// TIA Portal V19 export
FUNCTION_BLOCK "TYPIC_C403_SF_LVE"   // FB131, FBD
TITLE = TYPIC_C403_SF_LVE: Detectiepunt
{ S7_Optimized_Access := 'TRUE' }
AUTHOR : OCOTECH
FAMILY : Typical
NAME : C403.802
// Logisch Object Besturing: C403.802
// 
// De subfunctie detectiepunt verzorgt de bediening en sturing van een SOSodetectiepunt vanuit 3B en is tevens het raakvlak tussen 3B en de interne sturing van het detectiepunt.
// stored: MemoryReserve 10, SetENOAutomatically false
   VAR_INPUT
      CFG_STR { ExternalAccessible := 'False'; ExternalVisible := 'False'; ExternalWritable := 'False'} : USInt;   // Nummer van de rijstrook (1 = rechterrijstrook)
      CFG_NUM { ExternalAccessible := 'False'; ExternalVisible := 'False'; ExternalWritable := 'False'} : Int;   // Nummer van het detectiepunt op de rijstrook volgens rijrichting
      CFG_POS1 { ExternalAccessible := 'False'; ExternalVisible := 'False'; ExternalWritable := 'False'} : USInt;   // FO-naam van de verkeerskoker (of op- / afrit) waar het detectiepunt staat
      CFG_POS2 { ExternalAccessible := 'False'; ExternalVisible := 'False'; ExternalWritable := 'False'} : Real;   // Lengtepositie van het detectiepunt in de verkeerskoker
      CFG_LCK_AANT { ExternalAccessible := 'False'; ExternalVisible := 'False'; ExternalWritable := 'False'} : Int;   // Aantal stroomopwaartse detectiepunten waarin verkeerskundige meldingen onderdrukt worden
      STU_ALG_LCK_SIG { ExternalAccessible := 'False'; ExternalVisible := 'False'; ExternalWritable := 'False'} : USInt;   // Onderdruk alarmen
   END_VAR
   VAR_OUTPUT
      VAR_LVE { ExternalAccessible := 'False'; ExternalVisible := 'False'; ExternalWritable := 'False'} : "C403_VAR_LVE_TYPIC";   // Struct met alle variabelen van de SOS-sectie
   END_VAR
   VAR_IN_OUT
      STU_LVE : "C403_STU_LVE_TYPIC";   // Sturing Detectiepunten
      VAR_IF_LVE : "C403_VAR_IF_LVE_TYPIC";   // Struct met alle variabelen ontvangen van de functie (IF) in de interne sturing van het afsluitsysteem
   END_VAR
   VAR
      BED : Struct   // Bedieningen
         OBS : Struct   // SOS-sectie aan- of uitschakelen
            X : "UDT_BED_ALG";
            KNOP { S7_SetPoint := 'True'} : Array[0..1] of "UDT_BED_KNOP";
         END_STRUCT;
         VGV_SIG : Struct   // Signalering verkeerskundige alarmen vrijgeven of onderdrukken
            X : "UDT_BED_ALG";
            KNOP { S7_SetPoint := 'True'} : Array[0..1] of "UDT_BED_KNOP";
         END_STRUCT;
      END_STRUCT;
      BED_OBS { ExternalWritable := 'False'} : "TYPIC_HF_BED_ALG_KNOP";   // SOS-sectie aan- of uitschakelen
      BED_VGV_SIG { ExternalWritable := 'False'} : "TYPIC_HF_BED_ALG_KNOP";   // Signalering verkeerskundige alarmen vrijgeven of onderdrukken
      SIG { ExternalWritable := 'False'} : Struct   // Signaleringen
         AA01 : Bool;   // Detectiepunt niet observeerbaar
         AA02 : Bool;   // Storing algemeen
         AA03 : Bool;   // Deur wegkantkast geopend
         AV01 : Bool;   // Stilstand gedetecteerd
         AV02 : Bool;   // Snelheidsonderschrijding gedetecteerd
         AV03 : Bool;   // Spookrijder gedetecteerd
         A001 : Bool;   // Beveiliging aangesproken
         A002 : Bool;   // Storing detectiepunt
         A003 : Bool;   // Beveiliging klimaatregeling wegkantkast aangesproken
         A004 : Bool;   // Overspanningsbeveiliging aangesproken
      END_STRUCT;
      VAR { ExternalWritable := 'False'} : Struct   // Variabelen
         STS_STOP : USInt;   // Stilstand gedetecteerd
         STS_SOS : USInt;   // Snelheidsonderschrijding gedetecteerd
         RNO : USInt;   // Reden niet bestuurbaar
         VGV_SIG_VOP : Bool;   // TRUE = Signaleringen vrijgegeven voor verkeersoperator FALSE = Onderdrukt
         MEM_STS_STOP { ExternalAccessible := 'False'; ExternalVisible := 'False'} : Bool;   // TRUE = Stilstand gedetecteerd
         MEM_STS_SOS { ExternalAccessible := 'False'; ExternalVisible := 'False'} : Bool;   // TRUE = Snelheidsonderschrijding gedetecteerd
         STS_STOP_NEW { ExternalAccessible := 'False'; ExternalVisible := 'False'} : Bool;   // TRUE = Nieuwe detectie Stilstand
         STS_SOS_NEW { ExternalAccessible := 'False'; ExternalVisible := 'False'} : Bool;   // TRUE = Nieuwe detectie snelheidsonderschrijding
         LCK_STOP { ExternalAccessible := 'False'; ExternalVisible := 'False'} : Bool;   // TRUE = Onderdrukken signalering stilstand
         LCK_SOS { ExternalAccessible := 'False'; ExternalVisible := 'False'} : Bool;   // TRUE = Onderdrukken signalering SOS
         BSC : USInt;   // Beschikbaarheid
         STS_NEG : USInt;   // Spookrijder gedetecteerd
         OBS { ExternalAccessible := 'False'; ExternalVisible := 'False'} : USInt;   // Observeerbaarheid
         SIG_AV01 { ExternalAccessible := 'False'; ExternalVisible := 'False'} : USInt;   // Signalering Stilstand gedetecteerd actief
         SIG_AV02 { ExternalAccessible := 'False'; ExternalVisible := 'False'} : USInt;   // Signalering Snelheidsonderschrijding actief
         POS { ExternalAccessible := 'False'; ExternalVisible := 'False'} : Bool;   // Positie van het detectiepunt
      END_STRUCT;
      HF_BST_OBS { ExternalAccessible := 'False'; ExternalVisible := 'False'; ExternalWritable := 'False'} : "TYPIC_HF_BST_OBS";   // Hulp functie besturing
   END_VAR
   // // BED.OBS.KNOP[0] : InDienst
   // // BED.OBS.KNOP[1] : UitDienst
   // // BED.VGV_SIG.KNOP[0] : Ja
   // // BED.VGV_SIG.KNOP[1] : Onderdrukt
BEGIN

REGION Network 1: START
END_REGION

REGION Network 2: +++ Bedieningen +++
   // Vrijgave en verwerking van de bedieningen (centrale en lokale bediening). De bedienwaardes worden daarna in de verdere deelfunctionaliteiten gebruikt.
END_REGION

REGION Network 3: Knoppen BED_OBS(SOS-sectie aan- of uitschakelen)
   // Waardes en vrijge van de knoppen BED_OBS
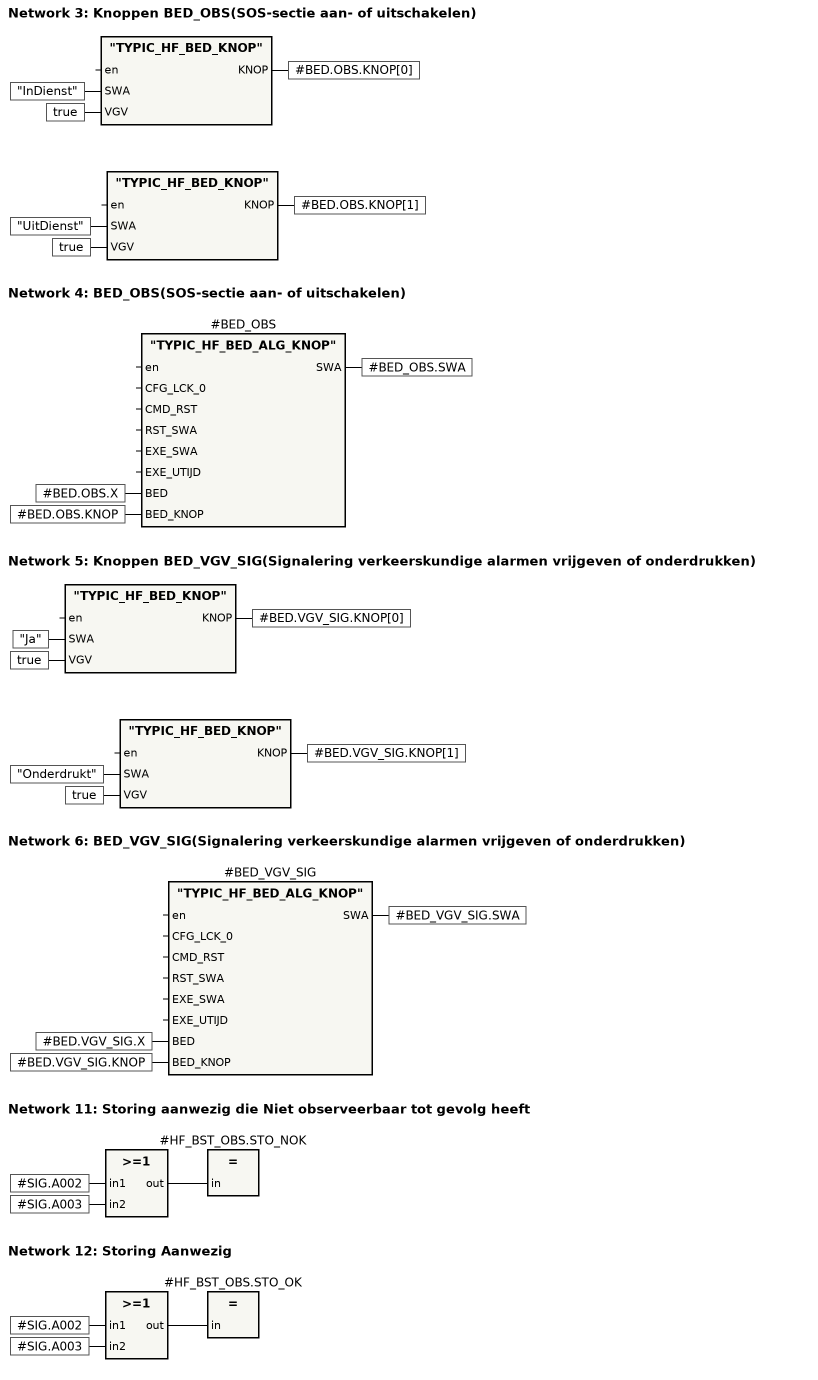
   "TYPIC_HF_BED_KNOP"(SWA := "InDienst", VGV := true, KNOP => #BED.OBS.KNOP[0]);
   "TYPIC_HF_BED_KNOP"(SWA := "UitDienst", VGV := true, KNOP => #BED.OBS.KNOP[1]);
END_REGION

REGION Network 4: BED_OBS(SOS-sectie aan- of uitschakelen)
   // Verwerking BED_OBS
   #BED_OBS(BED := #BED.OBS.X, BED_KNOP := #BED.OBS.KNOP, SWA => #BED_OBS.SWA);   // "TYPIC_HF_BED_ALG_KNOP"
END_REGION

REGION Network 5: Knoppen BED_VGV_SIG(Signalering verkeerskundige alarmen vrijgeven of onderdrukken)
   // Waardes en vrijge van de knoppen BED_VGV_SIG
   "TYPIC_HF_BED_KNOP"(SWA := "Ja", VGV := true, KNOP => #BED.VGV_SIG.KNOP[0]);
   "TYPIC_HF_BED_KNOP"(SWA := "Onderdrukt", VGV := true, KNOP => #BED.VGV_SIG.KNOP[1]);
END_REGION

REGION Network 6: BED_VGV_SIG(Signalering verkeerskundige alarmen vrijgeven of onderdrukken)
   // Verwerking BED_VGV_SIG
   #BED_VGV_SIG(BED := #BED.VGV_SIG.X, BED_KNOP := #BED.VGV_SIG.KNOP, SWA => #BED_VGV_SIG.SWA);   // "TYPIC_HF_BED_ALG_KNOP"
END_REGION

REGION Network 7: +++ Verwerken verkeersstatus +++
   // De ontvangen verkeersstatus vanuit de interne sturing omzetten naar variabelen
END_REGION

REGION Network 8: +++ Voorwaarden signalering stilstand +++
   // Een stilstand wordt gesignaleerd als bij opkomen van de detectie stilstand er geen onderdrukking is. Signaleringen kunnen onderdrukt worden als er detectiepunten stroomafwaarts reeds een stilstand signaleren.
END_REGION

REGION Network 9: +++ Voorwaarden signalering snelheidsonderschrijding +++
   // Een snelheidsonderschrijding wordt gesignaleerd als bij opkomen van de detectie snelheidsonderschrijding er geen onderdrukking is. Signaleringen kunnen onderdrukt worden als er detectiepunten stroomafwaarts reeds een snelheidsonderschrijding signaleren.
END_REGION

REGION Network 10: +++ Signaleringen en observeerbaarheid +++
   // Aanmaken signaleringen, bepalen observeerbaarheid (observeerbaar / niet observeerbaar) en bepalen reden niet observeerbaar.
END_REGION

REGION Network 11: Storing aanwezig die Niet observeerbaar tot gevolg heeft
   // OR-verknoping van alle storingen om input STO_BST_NOK van de hulpfunctie "Observeerbaarheid en algemene signlaring"
   #HF_BST_OBS.STO_NOK := #SIG.A002 OR #SIG.A003;
END_REGION

REGION Network 12: Storing Aanwezig
   // OR-verknoping van alle storingen om input STO_BST_OK van de hulpfunctie "Observeerbaarheid en algemene signlaring"
   #HF_BST_OBS.STO_OK := #SIG.A002 OR #SIG.A003;
END_REGION

REGION Network 13: Hulpfunctie "Observeerbaarheid en algemene signalering "
   // Bepalen variabele "Observeerbaarheid" en "reden niet Observeerbaarheid", Signaleringen "Observeerbaarheid" en "algmene storing".
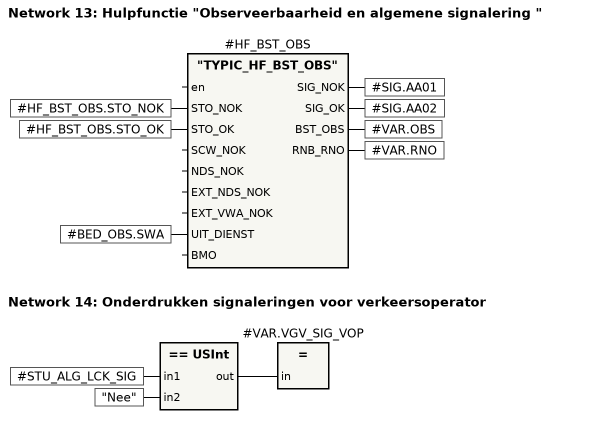
   #HF_BST_OBS(STO_NOK := #HF_BST_OBS.STO_NOK,   // "TYPIC_HF_BST_OBS"
               STO_OK := #HF_BST_OBS.STO_OK,
               UIT_DIENST := #BED_OBS.SWA,
               SIG_NOK => #SIG.AA01,
               SIG_OK => #SIG.AA02,
               BST_OBS => #VAR.OBS,
               RNB_RNO => #VAR.RNO);
END_REGION

REGION Network 14: Onderdrukken signaleringen voor verkeersoperator
   // Via de variabele VGV_SIG_VOP wordt aan IRIS SCADA doorgegeven of signaleringen (bestemd voor de verkeersoperator) van de deze functie zichtbaar (of onderdrukt) moeten zijn.
   #VAR.VGV_SIG_VOP := #STU_ALG_LCK_SIG = "Nee";
END_REGION

REGION Network 15: +++ Bepalen beschikbaarheidsstatus +++
   // Beschikbaarheidsstatus (Uit Dienst / beschikbaar / beperkt beschikbaar / niet beschikbaar) bepalen.
END_REGION

REGION Network 16 (SCL): Beschikbaarheidsstatus bepalen
   IF 
       //voorwaarden "Niet beschikbaar"
       TRUE
   THEN
       //Beschikbaarheidsstatus = Niet Beschikbaar
       #VAR.BSC:= "NietBeschikbaar";
   ELSIF
       //voorwaarden "Beperkt beschikbaar"
       TRUE
   THEN
       //Beschikbaarheidsstatus = Beperkt Beschikbaar
       #VAR.BSC:= "Beperkt";
   ELSE
       //Beschikbaarheidsstatus = Beschikbaar
       #VAR.BSC:= "Beschikbaar";
   END_IF;
END_REGION

REGION Network 17: +++ Verwerken configuraties +++
   // De configuraties verwerken naar variabelen.
END_REGION

REGION Network 18 (SCL): EINDE
   // Variabelen van intern scada rakvlak naar outputs copieren
   #VAR_LVE.BSC := #VAR.BSC;
   #VAR_LVE.STS_NEG := #VAR.STS_NEG;
   #VAR_LVE.OBS := #VAR.OBS;
   #VAR_LVE.SIG_AV01 := #VAR.SIG_AV01;
   #VAR_LVE.SIG_AV02 := #VAR.SIG_AV02;
   #VAR_LVE.POS := #VAR.POS;
END_REGION
END_FUNCTION_BLOCK
